{attribute addProperty BoxType "EP3182-1002-0017"}
{attribute addProperty Id "AI_Standard_ChannelAT %I*ARRAY[0..1] OF AI_Standard_Channel_5763EEB96480DO_OutputsAT %Q*DO_Outputs_E89552221620WcStateAT %I*WcState_98A4DF7520.250InfoDataAT %I*InfoData_BC63D37F80100"}
{attribute addProperty CRC "988524140"}
{attribute addProperty SizeInBites "162"}
{attribute addProperty SizeInBytes "20.25"}
TYPE EP3182_12747D8E :
STRUCT
	{attribute addProperty Name "AI_Standard_Channel"}
	AI_Standard_Channel : ARRAY[0..1] OF AI_Standard_Channel_5763EEB9;
	{attribute addProperty Name "DO_Outputs"}
	DO_Outputs : DO_Outputs_E8955222;
	{attribute addProperty Name "WcState"}
	WcState : WcState_98A4DF75;
	{attribute addProperty Name "InfoData"}
	InfoData : InfoData_BC63D37F;
END_STRUCT
END_TYPE

(* stored: Version 1.2.0.0, ProductVersion 3.1.4024.9
   DUT EP3182_12747D8E: Id {e74eebe5-82f7-466e-b107-98d59fc65869} *)
